FUNCTION_BLOCK RESET_M (* Composite Function Block Type *)
  (* Standard: 61499-2 *)
  (* Version 1.0, 2019-04-05, adeel *)
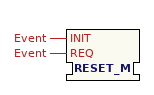
  EVENT_INPUT
    INIT;
    REQ; (* Normal Execution Request *)
  END_EVENT
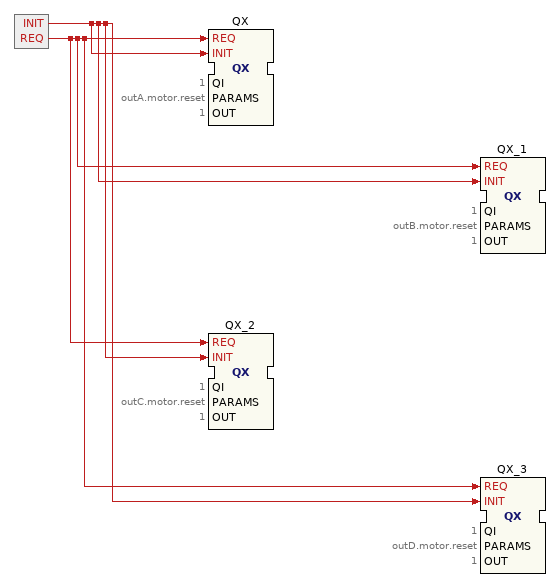
  FBS
    QX : QX(QI := 1, PARAMS := outA.motor.reset, OUT := 1);
    QX_1 : QX(QI := 1, PARAMS := outB.motor.reset, OUT := 1);
    QX_2 : QX(QI := 1, PARAMS := outC.motor.reset, OUT := 1);
    QX_3 : QX(QI := 1, PARAMS := outD.motor.reset, OUT := 1);
  END_FBS
  EVENT_CONNECTIONS
    REQ TO QX.REQ;
    REQ TO QX_2.REQ;
    REQ TO QX_1.REQ;
    REQ TO QX_3.REQ;
    INIT TO QX.INIT;
    INIT TO QX_1.INIT;
    INIT TO QX_2.INIT;
    INIT TO QX_3.INIT;
  END_CONNECTIONS
END_FUNCTION_BLOCK
